// TIA Portal V17 export
// export: Created 2022-07-20T07:02:42.2188255Z, ExportSetting WithDefaults, DisplayName Totally Integrated Automation Portal, DisplayVersion V17, DisplayName TIA Portal Openness, DisplayVersion V17, DisplayName TIA Portal Version Control Interface, DisplayVersion V17, DisplayName SINAMICS Startdrive Advanced, DisplayVersion V17, DisplayName SINAMICS Startdrive G130, G150, S120, S150, SINAMICS MV, S210, DisplayVersion V17, DisplayName SINAMICS Startdrive G110M, G120, G120C, G120D, G120P, G115D, DisplayVersion V17, DisplayName STEP 7 Professional, DisplayVersion V17, DisplayName STEP 7 Safety, DisplayVersion V17, DisplayName WinCC Advanced, DisplayVersion V17
DATA_BLOCK "InstCtrlHscExt"   // DB2
// stored: AutoNumber true, DBAccessibleFromOPCUA true, InstanceOfName HSC, OfSystemLibElement CTRL_HSC_EXT, OfSystemLibVersion 1.0
"HSC"
   // VAR_INPUT
   //    HSC : HW_HSC;
   // END_VAR
   // VAR_OUTPUT
   //    DONE : Bool;
   //    BUSY : Bool;
   //    ERROR : Bool;
   //    STATUS : Word;
   // END_VAR
   // VAR_IN_OUT
   //    CTRL : Variant;
   // END_VAR
BEGIN
END_DATA_BLOCK
